# EPICS autosave request: tomoScanApp/Db/tomoScan_PSO_settings.req
# This file is used by autosave to determine what PVs to save
# It is also used by tomoScan to determine what PVs to create

# This is the file for the TomoScanPSO derived class.

$(P)$(R)PSOPulseWidth
#controlPV $(P)$(R)PSOControllerModel
#controlPV $(P)$(R)PSOEncoderCountsPerStep
#controlPV $(P)$(R)PSOAxisName
#controlPV $(P)$(R)PSOEncoderInput
#controlPV $(P)$(R)PSOCountsPerRotation
#controlPV $(P)$(R)PSOStartTaxi
#controlPV $(P)$(R)PSOEndTaxi
#controlPV $(P)$(R)PSOCommand.BOUT
#controlPV $(P)$(R)PSOCommand.BINP
$(P)$(R)ProgramPSO
